(* CoDeSys 2.3 library: Ethernet.lib *)

(* Global variable list: CONST_ETHERNET_LIB *)
VAR_GLOBAL CONSTANT
	(*--- ETH_ERRORS ---------------------------------------------------------------------------------------------------------------*)
	NO_ERROR					:	WORD :=16#0000; 	(* no error *)
	FNC_NOT_SUPPORTED		:	WORD :=16#0001;	(*the function is not supported by the firmware *)
	EIO							:	WORD :=16#8001;	(* Input/output error *)
	ENXIO							:	WORD :=16#8002;	(* Device not configured *)
	EINVAL						:	WORD :=16#8003;	(* Invalid argument *)
	EALREADY					:	WORD :=16#8004;	(* Operation already in progress *)
	EDESTADDRREQ			:	WORD :=16#8005;	(* Destination address required *)
	EMSGSIZE					:	WORD :=16#8006;	(* Message too long *)
	EPROTOTYPE				:	WORD :=16#8007;	(* Protocol wrong type for socket *)
	ENOPROTOOPT				:	WORD :=16#8008;	(* Protocol not available *)
	EPROTONOSUPPORT		:	WORD :=16#8009;	(* Protocol not supported *)
	ESOCKTNOSUPPORT		:	WORD :=16#800A;	(* Socket type not supported *)
	EOPNOTSUPP				:	WORD :=16#800B;	(* Operation not supported *)
	EAFNOSUPPORT				:	WORD :=16#800C;	(* Address family not supported by protocol family *)
	EADDRINUSE					:	WORD :=16#800D;	(* Address already in use *)
	EADDRNOTAVAIL				:	WORD :=16#800E;	(* Can't assign requested address *)
	ENETDOWN					:	WORD :=16#800F;	(* Network is down *)
	ENETUNREACH				:	WORD :=16#8010;	(* Network is unreachable *)
	ENETRESET					:	WORD :=16#8011;	(* Network dropped connection on reset *)
	ECONNABORTED			:	WORD :=16#8012;	(* Software caused connection abort *)
	ECONNRESET				:	WORD :=16#8013;	(* Connection reset by peer *)
	ENOBUFS						:	WORD :=16#8014;	(* No buffer space available *)
	EISCONN						:	WORD :=16#8015;	(* Socket is already connected *)
	ENOTCONN					:	WORD :=16#8016;	(* Socket is not connected *)
	ESHUTDOWN					:	WORD :=16#8017;	(* Can't send after socket shutdown *)
	ETIMEDOUT					:	WORD :=16#8018;	(* Operation timed out *)
	ECONNREFUSED			:	WORD :=16#8019;	(* Connection refused *)
	EHOSTDOWN					:	WORD :=16#801A;	(* Host is down *)
	EHOSTUNREACH			:	WORD :=16#801B;	(* No route to host *)
	EACCES						:	WORD :=16#801C;  	(* access permision *)
	ESRCH						:	WORD :=16#801D;  	(* search failed *)
	EEXIST						:	WORD :=16#801E;	(* route exists previously *)
	EPIPE							:	WORD :=16#801F;	(* broken communication channel *)
	EWOULDBLOCK				:	WORD :=16#8020; 	(* communication should be blocking *)
	ETOOMANYREFS				:	WORD :=16#8021;  	(* number of maximal multicast members reached *)
	EDOM							:	WORD :=16#8022; 	(* value exceeds domain *)
	ENOREF						:	WORD :=16#8023; 	(* no reference to socket *)
	SOCKAPI_NODESCRIPTOR	:	WORD :=16#C001; 	(* no free socket descriptor for this open call *)
	SOCKAPI_INVALID_IP		:	WORD :=16#C002; 	(* Trying to configure an invalid IP address *)
	(*------------------------------------------------------------------------------------------------------------------------------------------------*)



END_VAR

(* Data type *)
TYPE ETH_ERROR : WORD;
END_TYPE

(* For possible ETH_ERROR values please see CONST_ETHERNET_LIB in the global var section *)

(* Data type *)
TYPE SEL_PROTOCOL :(
	IPPROTO_IP 		:= 0,		(* dummy FOR IP *)
	IPPROTO_ICMP 	:= 1,		(* control message protocol *)
	IPPROTO_IGMP 	:= 2,		(* group mgmt protocol *)
	IPPROTO_TCP 	:= 6,		(* tcp *)
	IPPROTO_UDP 	:= 17,		(* user datagram protocol *)
	IPPROTO_RAW 	:= 255);	(* raw IP packet *)
END_TYPE

(* Data type *)
TYPE SEL_TYPE :(
	SOCK_STREAM 	:=1,		(* stream socket *)
	SOCK_DGRAM 	:=	2,		(* datagram socket *)
	SOCK_RAW 		:=	3);		(* raw-protocol interface *)
END_TYPE

(* POU ETHERNET_CLIENT_CLOSE, IL *)
FUNCTIONBLOCK ETHERNET_CLIENT_CLOSE (* close a client socket *)

VAR_INPUT
	EN			:	BOOL;
	SOCKET	:	WORD;
END_VAR

VAR_OUTPUT
	ENO		:	BOOL;
	ERROR	:	ETH_ERROR;
END_VAR
LD	0
END_FUNCTION_BLOCK

(* POU ETHERNET_CLIENT_OPEN, IL *)
FUNCTIONBLOCK ETHERNET_CLIENT_OPEN (* open a socket *)

VAR_INPUT
	EN			:	BOOL;
	TYP		:	SEL_TYPE;
	PROTO	:	SEL_PROTOCOL;
	IP_ADR	:	DWORD;
	PORT		:	WORD;
END_VAR

VAR_OUTPUT
	ENO		:	BOOL;
	SOCKET	:	WORD;
	ERROR	:	ETH_ERROR;
END_VAR

VAR
	AUX		:	BOOL;
END_VAR
LD	0
END_FUNCTION_BLOCK

(* POU ETHERNET_GET_NETWORK_CONFIG, IL *)
FUNCTIONBLOCK ETHERNET_GET_NETWORK_CONFIG (* get Network configuration *)

VAR_INPUT
	EN					:	BOOL;
END_VAR

VAR_OUTPUT
	ENO				:	BOOL;
	IP_ADR			:	DWORD;
	GW_ADR			:	DWORD;
	SUBNET_MASK	:	DWORD;
END_VAR
LD	0
END_FUNCTION_BLOCK

(* POU ETHERNET_READ, IL *)
FUNCTIONBLOCK ETHERNET_READ (* read data *)

VAR_INPUT
	EN				:	BOOL;
	SOCKET		:	WORD;
END_VAR

VAR_OUTPUT
	ENO			:	BOOL;
	ERROR		:	ETH_ERROR;
	LEN_OUT		:	WORD;
	SRC_IP		:	DWORD;
	SRC_PORT	:	WORD;
END_VAR

VAR_IN_OUT
	DATA			:	ARRAY [1 .. 1500] OF  BYTE;
END_VAR
LD	0
END_FUNCTION_BLOCK

(* POU ETHERNET_READ_PT, IL *)
FUNCTIONBLOCK ETHERNET_READ_PT (* read data *)

VAR_INPUT
	EN				:	BOOL;
	SOCKET		:	WORD;
END_VAR

VAR_OUTPUT
	ENO			:	BOOL;
	ERROR		:	ETH_ERROR;
	LEN_OUT		:	WORD;
	SRC_IP		:	DWORD;
	SRC_PORT	:	WORD;
END_VAR

VAR_IN_OUT
	DATA_PT		:	POINTER TO ARRAY [1 .. 1500] OF  BYTE;
END_VAR
LD	0
END_FUNCTION_BLOCK

(* POU ETHERNET_SERVER_OPEN, IL *)
FUNCTIONBLOCK ETHERNET_SERVER_OPEN (* open a socket *)

VAR_INPUT
	EN			:	BOOL;
	TYP		:	SEL_TYPE;
	PROTO	:	SEL_PROTOCOL;
	PORT		:	WORD;
END_VAR

VAR_OUTPUT
	ENO		:	BOOL;
	SOCKET	:	WORD;
	ERROR	:	ETH_ERROR;
END_VAR
LD	0
END_FUNCTION_BLOCK

(* POU ETHERNET_SET_NETWORK_CONFIG, IL *)
FUNCTIONBLOCK ETHERNET_SET_NETWORK_CONFIG (* get IP addresst *)

VAR_INPUT
	EN					:	BOOL;
	IP_ADR			:	DWORD;
	GW_ADR			:	DWORD;
	SUBNET_MASK	:	DWORD;
END_VAR

VAR_OUTPUT
	ENO				:	BOOL;
	ERROR			:	ETH_ERROR;
END_VAR
LD	0
END_FUNCTION_BLOCK

(* POU ETHERNET_WRITE, IL *)
FUNCTIONBLOCK ETHERNET_WRITE (* write data  *)

VAR_INPUT
	EN				:	BOOL;
	SOCKET		:	WORD;
	LEN_IN		:	WORD;
	DST_IP		:	DWORD;
	DST_PORT	:	WORD;
END_VAR

VAR_OUTPUT
	ENO			:	BOOL;
	ERROR		:	ETH_ERROR;
END_VAR

VAR_IN_OUT
	DATA			:	ARRAY [1 .. 1500] OF  BYTE;
END_VAR
LD	0
END_FUNCTION_BLOCK

(* POU ETHERNET_WRITE_PT, IL *)
FUNCTIONBLOCK ETHERNET_WRITE_PT (* write data  *)

VAR_INPUT
	EN				:	BOOL;
	SOCKET		:	WORD;
	LEN_IN		:	WORD;
	DST_IP		:	DWORD;
	DST_PORT	:	WORD;
END_VAR

VAR_OUTPUT
	ENO			:	BOOL;
	ERROR		:	ETH_ERROR;
END_VAR

VAR_IN_OUT
	DATA_PT		:	POINTER TO ARRAY [1 .. 1500] OF  BYTE;
END_VAR
	LD		0
END_FUNCTION_BLOCK

(* POU ETHERNET_CLIENT_OPEN_2, IL *)
FUNCTION_BLOCK ETHERNET_CLIENT_OPEN_2

VAR_INPUT
	EN			:	BOOL;
	TYP		:	SEL_TYPE;
	PROTO	:	SEL_PROTOCOL;
	IP_ADR	:	DWORD;
	PORT		:	WORD;
      TIMEOUT	:	DWORD;  (* Timeout in ms *)
END_VAR

VAR_OUTPUT
	ENO		:	BOOL;
	SOCKET	:	WORD;
	ERROR	:	ETH_ERROR;
END_VAR

VAR
	AUX		:	BOOL;
END_VAR
	LD		0
END_FUNCTION_BLOCK

(* POU ETHERNET_GET_VARIABLES, IL *)
FUNCTION_BLOCK ETHERNET_GET_VARIABLES

VAR_INPUT
	EN						:	BOOL;
END_VAR

VAR_OUTPUT
	BootpRequest			:	WORD;
	ConnectionWdTime	:	WORD;
	ENO					:	BOOL;
	ERROR				:	ETH_ERROR;
END_VAR

VAR
END_VAR
LD 0
END_FUNCTION_BLOCK

(* POU ETHERNET_GETSOURCEPORT, IL *)
FUNCTION_BLOCK ETHERNET_GETSOURCEPORT

VAR_INPUT
	EN			:	BOOL;
	SOCKET	:	WORD;
END_VAR

VAR_OUTPUT
	SPORT	:	WORD;
	ENO		:	BOOL;
	ERROR	:	ETH_ERROR;
END_VAR

VAR
END_VAR
LD 0
END_FUNCTION_BLOCK

(* POU ETHERNET_SERVER_CLOSE, IL *)
FUNCTION_BLOCK ETHERNET_SERVER_CLOSE (* close a server socket *)

VAR_INPUT
	EN			:	BOOL;
	SOCKET	:	WORD;
END_VAR

VAR_OUTPUT
	ENO		:	BOOL;
	ERROR	:	ETH_ERROR;
END_VAR
LD 0
END_FUNCTION_BLOCK

(* POU ETHERNET_SET_VARIABLES, IL *)
FUNCTION_BLOCK ETHERNET_SET_VARIABLES

VAR_INPUT
	EN						:	BOOL;
	BootpRequest			:	WORD;
	ConnectionWdTime	:	WORD;
END_VAR

VAR_OUTPUT
	ENO					:	BOOL;
	ERROR				:	ETH_ERROR;
END_VAR

VAR
END_VAR
LD 0
END_FUNCTION_BLOCK

(* POU ETHERNET_SETSOURCEPORT, IL *)
FUNCTION_BLOCK ETHERNET_SETSOURCEPORT

VAR_INPUT
	EN			:	BOOL;
	SOCKET	:	WORD;
	SPORT	:	WORD;
END_VAR

VAR_OUTPUT
	ENO		:	BOOL;
	ERROR	:	ETH_ERROR;
END_VAR

VAR
END_VAR
LD 0
END_FUNCTION_BLOCK

(* POU ETHERNET_VERSION, IL *)
FUNCTION ETHERNET_VERSION : WORD

VAR_INPUT
	EN	: BOOL;
END_VAR
LD 0
END_FUNCTION
